FUNCTION_BLOCK FB_ActuatorDecoratorTest EXTENDS FB_BaseControlElementDecoratorParent IMPLEMENTS ITF_ActuatorDecoratorTest
VAR
	itfactActuator		: ITF_Actuator;
	itfsenStart			: ITF_SensorDecoratorTest;
	itfsenEnd			: ITF_SensorDecoratorTest;
	
END_VAR

METHOD FB_init : BOOL
VAR_INPUT
	bInitRetains : BOOL; // if TRUE, the retain variables are initialized (warm start / cold start)
	bInCopyCode : BOOL;  // if TRUE, the instance afterwards gets moved into the copy code (online change)
	fbToDecorate		: ITF_DecoratedElement;
	actActuator			: ITF_Actuator;
	senStart			: ITF_SensorDecoratorTest;
	senEnd				: ITF_SensorDecoratorTest;
	
END_VAR
THIS^.itfactActuator	:= actActuator;
THIS^.itfsenStart		:= senStart;
THIS^.itfsenEnd			:= senEnd;
END_METHOD

METHOD IsEnd : BOOL
VAR_INPUT
END_VAR
IsEnd		:= THIS^.itfactActuator.IsEnd ();
END_METHOD

METHOD PUBLIC IsStart : BOOL
VAR_INPUT
END_VAR
IsStart		:= THIS^.itfactActuator.IsStart ();
END_METHOD

(*			
	EVERDE sp. z o.o.
	Rafał Osajda		31.03.2025		TC 4024.66
	Uruchomienie cyklu przesuwania do początku
*)
METHOD PUBLIC MoveToEnd
VAR_INPUT
END_VAR
THIS^.itfactActuator.MoveToEnd ();
END_METHOD

(*			
	EVERDE sp. z o.o.
	Rafał Osajda		31.03.2025		TC 4024.66
	Uruchomienie cyklu przesuwania do początku
*)
METHOD PUBLIC MoveToStart
VAR_INPUT
END_VAR
THIS^.itfactActuator.MoveToStart ();
END_METHOD

METHOD PUBLIC MovingToEndBusy : BOOL
VAR_INPUT
END_VAR
MovingToEndBusy		:= THIS^.itfactActuator.MovingToEndBusy ();
END_METHOD

METHOD PUBLIC MovingToEndFirstCycyle : BOOL
VAR_INPUT
END_VAR
MovingToEndFirstCycyle		:= THIS^.itfactActuator.MovingToEndFirstCycyle ();
END_METHOD

METHOD PUBLIC MovingToEndStatus : BOOL
VAR_INPUT
END_VAR
MovingToEndStatus		:= THIS^.itfactActuator.MovingToEndStatus ();
END_METHOD

METHOD PUBLIC MovingToStartBusy : BOOL
VAR_INPUT
END_VAR
MovingToStartBusy		:= THIS^.itfactActuator.MovingToStartBusy ();
END_METHOD

METHOD PUBLIC MovingToStartFirstCycle : BOOL
VAR_INPUT
END_VAR
MovingToStartFirstCycle 	:= THIS^.itfactActuator.MovingToStartFirstCycle ();
END_METHOD

METHOD PUBLIC MovingToStartStatus : BOOL
VAR_INPUT
END_VAR
MovingToStartStatus		:= THIS^.itfactActuator.MovingToStartStatus ();
END_METHOD

END_FUNCTION_BLOCK

(* stored: Version 1.1.0.1
   POU FB_ActuatorDecoratorTest: Id {afef5ecf-7924-00e5-278c-76059101fe57}, SpecialFunc None
   Method FB_init: Id {33b0cda0-2287-032f-0727-14b915c1f328}
   Method IsEnd: Id {cec0f738-fc1c-0e8d-1394-63230a70e165}
   Method IsStart: Id {64260bb7-d289-0965-2999-708e3e909685}
   Method MoveToEnd: Id {642c8f48-fa3a-40fd-905f-d5deb33e924b}
   Method MoveToStart: Id {69e4a550-995f-4b44-9a57-c902d1d329c4}
   Method MovingToEndBusy: Id {ffa00487-3f69-4a75-99ea-b6dceb87f958}
   Method MovingToEndFirstCycyle: Id {195fd51a-1f9e-439d-b6ca-7878a6503b07}
   Method MovingToEndStatus: Id {82a57ba5-2422-4866-9fea-4c4e9d99d757}
   Method MovingToStartBusy: Id {19be314e-4c12-483e-9b8e-79d1d96c05a5}
   Method MovingToStartFirstCycle: Id {4327d628-239f-403d-b9c9-39318b88bdae}
   Method MovingToStartStatus: Id {48cfa4d0-18f2-437c-a350-fa507fff15ea} *)
